// TIA Portal V18 export
DATA_BLOCK "webData"   // DB8
{ S7_Optimized_Access := 'TRUE' }
VERSION : 0.1
// stored: AutoNumber true, DBAccessibleFromOPCUA true, DBAccessibleFromWebserver true, IsOnlyStoredInLoadMemory false, IsRetainMemResEnabled false, IsWriteProtectedInAS false, MemoryReserve 0
   VAR
      lineName { ExternalAccessible := 'False'; ExternalVisible := 'False'; ExternalWritable := 'False'} : WString := WSTRING#'L14';
      andon1Text { ExternalAccessible := 'False'; ExternalVisible := 'False'; ExternalWritable := 'False'} : WString := WSTRING#'Andon1';
      andon2Text { ExternalAccessible := 'False'; ExternalVisible := 'False'; ExternalWritable := 'False'} : WString := WSTRING#'Andon2';
      andon3Text { ExternalAccessible := 'False'; ExternalVisible := 'False'; ExternalWritable := 'False'} : WString := WSTRING#'Andon3';
      andon4Text { ExternalAccessible := 'False'; ExternalVisible := 'False'; ExternalWritable := 'False'} : WString := WSTRING#'Andon4';
      andon5Text { ExternalAccessible := 'False'; ExternalVisible := 'False'; ExternalWritable := 'False'} : WString := WSTRING#'Andon5';
      andon6Text { ExternalAccessible := 'False'; ExternalVisible := 'False'; ExternalWritable := 'False'} : WString := WSTRING#'Andon6';
      andon7Text { ExternalAccessible := 'False'; ExternalVisible := 'False'; ExternalWritable := 'False'} : WString := WSTRING#'Andon7';
      andon8Text { ExternalAccessible := 'False'; ExternalVisible := 'False'; ExternalWritable := 'False'} : WString := WSTRING#'Andon8';
      andon9Text { ExternalAccessible := 'False'; ExternalVisible := 'False'; ExternalWritable := 'False'} : WString := WSTRING#'Andon9';
      andon10Text { ExternalAccessible := 'False'; ExternalVisible := 'False'; ExternalWritable := 'False'} : WString := WSTRING#'Andon10';
      actualValues { ExternalAccessible := 'False'; ExternalVisible := 'False'; ExternalWritable := 'False'} : "UDT_actualValues";
      andon1state { ExternalAccessible := 'False'; ExternalVisible := 'False'; ExternalWritable := 'False'} : Int;
      andon2state { ExternalAccessible := 'False'; ExternalVisible := 'False'; ExternalWritable := 'False'} : Int;
      andon3state { ExternalAccessible := 'False'; ExternalVisible := 'False'; ExternalWritable := 'False'} : Int;
      andon4state { ExternalAccessible := 'False'; ExternalVisible := 'False'; ExternalWritable := 'False'} : Int;
      andon5state { ExternalAccessible := 'False'; ExternalVisible := 'False'; ExternalWritable := 'False'} : Int;
      andon6state { ExternalAccessible := 'False'; ExternalVisible := 'False'; ExternalWritable := 'False'} : Int;
      andon7state { ExternalAccessible := 'False'; ExternalVisible := 'False'; ExternalWritable := 'False'} : Int;
      andon8state { ExternalAccessible := 'False'; ExternalVisible := 'False'; ExternalWritable := 'False'} : Int;
      andon9state { ExternalAccessible := 'False'; ExternalVisible := 'False'; ExternalWritable := 'False'} : Int;
      andon10state { ExternalAccessible := 'False'; ExternalVisible := 'False'; ExternalWritable := 'False'} : Int;
   END_VAR
BEGIN
END_DATA_BLOCK
